# EPICS autosave request: ADRoper/roperApp/Db/roper_settings.req
$(P)$(R)NumAcquisitions
$(P)$(R)RoperShutterMode
$(P)$(R)AutoDataType
$(P)$(R)Temperature
$(P)$(R)Comment1
$(P)$(R)Comment2
$(P)$(R)Comment3
$(P)$(R)Comment4
$(P)$(R)Comment5
